(* CODESYS project Semaforo.project

Project tree, tasks and I/O mapping:
  Device : CODESYS Control Win V3, 3S - Smart Software Solutions GmbH, order no. 305021, version 3.5.10.30
    application Application
      libraries: Standard, * (System)
      task MainTask (cyclic, interval t#20ms, priority 1) calls PLC_PRG
      task VISU_TASK (cyclic, interval 100 ms, priority 31) calls VisuElems.Visu_Prg
      program PLC_PRG [FBD]
      function block NormalCycle [ST]
      function block BlinkingYellow [ST]
      visualisation Visualization
      function block Selettore [ST]
  text list GlobalTextList
*)

// Device/Application/PLC_PRG
PROGRAM PLC_PRG
VAR
	Red1: BOOL := FALSE;
	Red2: BOOL := FALSE;
	Red: BOOL;
	Yellow1: BOOL := FALSE;
	Yellow2: BOOL:= FALSE;
	Yellow: BOOL;
	Green1: BOOL := FALSE;
	Green2: BOOL := FALSE;
	Green: BOOL;
	NoermalCycle_0: NormalCycle;
	BlinkingYellow_0: BlinkingYellow;	
	Selettore_0: Selettore;
	TickErr: BOOL := FALSE;
	Channel: INT := 0;	
END_VAR

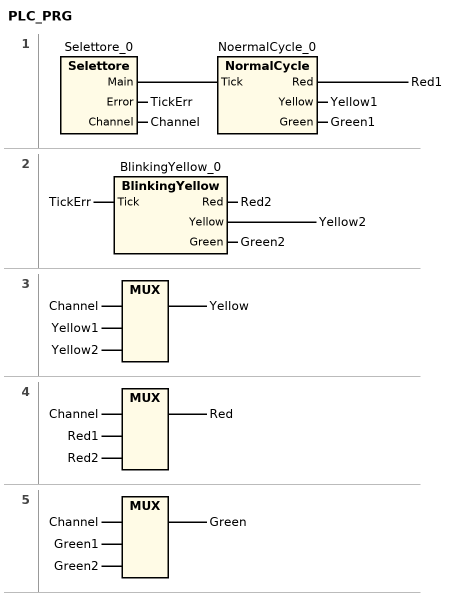
// NETWORK 1
Selettore_0(Error => TickErr, Channel => Channel); // Selettore
NoermalCycle_0(Tick := Selettore_0.Main, Yellow => Yellow1, Green => Green1); // NormalCycle
Red1 := NoermalCycle_0.Red;

// NETWORK 2
BlinkingYellow_0(Tick := TickErr, Red => Red2, Green => Green2); // BlinkingYellow
Yellow2 := BlinkingYellow_0.Yellow;

// NETWORK 3
Yellow := MUX(Channel, Yellow1, Yellow2);

// NETWORK 4
Red := MUX(Channel, Red1, Red2);

// NETWORK 5
Green := MUX(Channel, Green1, Green2);

END_PROGRAM

// Device/Application/NormalCycle
FUNCTION_BLOCK NormalCycle
VAR_OUTPUT
	Red: BOOL := FALSE;
	Yellow: BOOL := FALSE;
	Green: BOOL := FALSE;
END_VAR
VAR	
	CounterR: TIME := T#3S;
	CounterY: TIME := T#5S;
	CounterG: TIME := T#4S;
	count: INT := 0;	
	Wait: TON;
END_VAR

VAR_INPUT
	Tick: BOOL := FALSE;
END_VAR

IF Tick = TRUE THEN
	CASE count OF
	0:// Red   
		Red := TRUE;
		Green := FALSE;
     	Yellow := FALSE;
     
		wait(IN:=TRUE, PT:=CounterR);		
		IF wait.Q THEN
			wait(IN:=FALSE);
			count := count + 1;
		END_IF;
  	 1: // Green    		
   		Red := FALSE;
		Green := TRUE;
     	Yellow := FALSE;
     
     	wait(IN:=TRUE, PT:=CounterG);	
		IF wait.Q THEN
			wait(IN:=FALSE);
			count := count + 1;
		END_IF;
   	2:  // Green and Yellow
		Red := FALSE;
		Green := TRUE;
     	Yellow := TRUE;
     
     	wait(IN:=TRUE, PT:=CounterY);     		
     	IF wait.Q THEN
     		wait(IN:=FALSE);
     		count := count + 1;
     	END_IF;   		
		ELSE
		count := 0;
	END_CASE;
END_IF

END_FUNCTION_BLOCK

// Device/Application/Selettore
FUNCTION_BLOCK Selettore
VAR_OUTPUT
	Main: BOOL := FALSE;
	Error: BOOL := FALSE;
	Channel: INT := 0;
END_VAR
VAR
	Count : INT := 0;
	wait : TON;	
END_VAR

CASE count OF
	0: // On
			Main := TRUE;
			Error := FALSE;	
			Channel := 0;			
			wait(IN:=TRUE, PT:=T#24S);			
			IF wait.Q THEN
				wait(IN:=FALSE);
				count := count + 1;
			END_IF;	
	1: // Off
			Main := FALSE;
			Error := TRUE; 
			Channel := 1;  	  		
   				
END_CASE

END_FUNCTION_BLOCK

// Device/Application/BlinkingYellow
FUNCTION_BLOCK BlinkingYellow
VAR_OUTPUT	
	Red: BOOL := TRUE;
	Yellow: BOOL := FALSE;
	Green: BOOL := TRUE;
END_VAR
VAR_INPUT
	Tick: BOOL;
END_VAR
VAR
	count : INT := 0;
	Counter: TIME := T#3S;
	Wait: TON;	
	
END_VAR

IF Tick = TRUE THEN
	Red := FALSE;
	Yellow:= FALSE;
	Green := FALSE;
	
	CASE count OF
	0: // On	   
			Yellow := TRUE;			
			wait(IN:=TRUE, PT:=T#2S);
			
			IF wait.Q THEN
				wait(IN:=FALSE);
				count := count + 1;
			END_IF;	
	1: // Off
   
   		Yellow 	:= FALSE;   		
   		wait(IN:=TRUE, PT:=T#2S);
   		
   		IF wait.Q THEN
   			wait(IN:=FALSE);
   			count := 0;
   		END_IF;		
	END_CASE
END_IF

END_FUNCTION_BLOCK

// Device/Application/Visualization
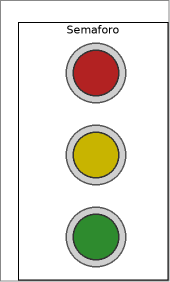
VISUALIZATION Visualization  // 170x282
    Rectangle (18,22 150x258), "Semaforo"
    Lamp1 (61,202 70x70), variable: PLC_PRG.Green, style: Lamp-Lamp1-Green
    Lamp1 (61,120 70x70), variable: PLC_PRG.Yellow, style: Lamp-Lamp1-Yellow
    Lamp1 (61,38 70x70), variable: PLC_PRG.Red, style: Lamp-Lamp1-Red
END_VISUALIZATION
